// TIA Portal V18 export
// export: Created 2026-06-08T05:50:11Z, ExportSetting WithDefaults
PlcWatchTable "WT_Test_Import_Schema"
  PlcWatchTableEntry "AI_MB_TCP_iStep"
  PlcWatchTableEntry "AI_MB_TCP_Write_Req"
